FUNCTION_BLOCK FB_SlaveRobot
VAR_INPUT
END_VAR
VAR_OUTPUT
END_VAR
VAR
	// flag if robot self-check passed
	m_selfCheckPass :ARRAY[1..g_sArmNum] OF BOOL :=[4(false)];
	
	// flag if master are connected
	m_masterOnLine :BOOL :=FALSE;
	m_masterOnLineCheck :FB_masterConnectionCheck;
	
	// master-slave motion scale
	m_motionScale :LREAL;
	
	// index(0 to 4) of slave arm which is tele-linked to master arm
	m_teleSlaveArmIdx :ARRAY[1..g_mArmNum] OF E_MatchedSlaveArmIdx;
	
	// flag if endoscope is mounted
	m_endoscopeMounted :BOOL := FALSE;
	
	// endoscope pose in cart coordinate
	m_endoscopePose : ST_Frame;
	
	// endoscope type 
	m_endoscopeType : E_EndoscopeType:= EndoScopeType_30;
	m_lastEndoScopePostureRobot : E_EndoscopePosture:= EndoScopePosture_HeadDown;
	m_lastEndoScopePostureUI : E_EndoscopePosture:= EndoScopePosture_HeadDown;
	
	// slave arms, responsible for arm kinematic and control
	m_slaveArms :ARRAY[1..g_sArmNum] OF FB_SlaveArm;
	
	// arm state
	m_slaveArmState:ARRAY[1..g_sArmNum] OF E_SlaveArmState:=[4(E_SlaveArmState.SlaveArmState_Error)];
	m_lastSlaveArmState:ARRAY[1..g_sArmNum] OF E_SlaveArmState:=[4(E_SlaveArmState.SlaveArmState_Error)];
	m_nextSlaveArmState:ARRAY[1..g_sArmNum] OF E_SlaveArmState:=[4(E_SlaveArmState.SlaveArmState_Error)];
	
	// matched master arm state
	m_matchedMasterArmState :ARRAY[1..g_sArmNum] OF E_MasterArmState:=[4(E_MasterArmState.MasterArmState_Error)];
	
	// flag if panel and instrument mounted
	m_panelMountedFlag :ARRAY[1..g_sArmNum] OF BOOL :=[4(FALSE)];
	m_instrumentMountedFlag :ARRAY[1..g_sArmNum] OF BOOL :=[4(FALSE)];
	
	// flag if enable instrument invasion after it mounted
	m_instruInvasionEnableFlag :ARRAY[1..g_sArmNum] OF BOOL :=[4(FALSE)];
	
	// all arm controller instance 
	m_armCtrlFactory :ARRAY[1..g_sArmNum,1..SlaveArmState_totalNum] OF I_SlaveArmCtrl;
	m_armError :ARRAY[1..g_sArmNum] OF FB_SlaveCtrlError;
	m_armInit :ARRAY[1..g_sArmNum] OF FB_SlaveCtrlInit;
	m_armSelfCheck :ARRAY[1..g_sArmNum] OF FB_SlaveCtrlSelfCheck;
	m_armStandBy :ARRAY[1..g_sArmNum] OF FB_SlaveCtrlStandBy;
	m_mountPanel :ARRAY[1..g_sArmNum] OF FB_SlaveCtrlMountPanel;
	m_panelReady :ARRAY[1..g_sArmNum] OF FB_SlaveCtrlPanelReady;
	m_mountInstru :ARRAY[1..g_sArmNum] OF FB_SlaveCtrlMountInstru;
	m_instruReady :ARRAY[1..g_sArmNum] OF FB_SlaveCtrlInstruReady;
	m_armMasterSlave :ARRAY[1..g_sArmNum] OF FB_SlaveCtrlMasterSlave;
	m_scopeReady :ARRAY[1..g_sArmNum] OF FB_SlaveCtrlScopeReady;
	m_armEndoscope :ARRAY[1..g_sArmNum] OF FB_SlaveCtrlEndoscope;
	m_armAdjust :ARRAY[1..g_sArmNum] OF FB_SlaveCtrlAdjust;
	m_armPackage :ARRAY[1..g_sArmNum] OF FB_SlaveCtrlPackage;
	m_armCart :ARRAY[1..g_sArmNum] OF FB_SlaveCtrlCart;
	m_armGraCali :ARRAY[1..g_sArmNum] OF FB_SlaveCtrlGraCali;
	m_armTest :ARRAY[1..g_sArmNum] OF FB_SlaveCtrlTest;
	m_instruRetract :ARRAY[1..g_sArmNum] OF FB_SlaveCtrlInstruRetract;
	m_instruInvasion :ARRAY[1..g_sArmNum] OF FB_SlaveCtrlInstruInvasion;
	m_armDisable :ARRAY[1..g_sArmNum] OF FB_SlaveCtrlDisable;
	m_instruCali :ARRAY[1..g_sArmNum] OF FB_SlaveCtrlInstruCali;
	m_scopeToggle :ARRAY[1..g_sArmNum] OF FB_SlaveCtrlScopeToggle;
	m_Performance :ARRAY[1..g_sArmNum] OF FB_SlaveCtrlPerformance;
	m_armStop :ARRAY[1..g_sArmNum] OF FB_SlaveCtrlStop;
	
	// arm controller interface
	m_armCtrl :ARRAY[1..g_sArmNum] OF I_SlaveArmCtrl;
	m_armCtrlCmds :ARRAY[1..g_sArmNum] OF ST_SlaveArmCtrlCmds;

END_VAR

METHOD PROTECTED controllerTransit : BOOL
VAR_INPUT
END_VAR
VAR
	i:int;
END_VAR
FOR i:=1 TO g_sArmNum DO 
	// Controller transit
	IF m_nextSlaveArmState[i]<> m_slaveArmState[i] THEN
		// reset current controller
		m_armCtrl[i].reset();
		
		// transit to new controller
		m_lastSlaveArmState[i]:=m_slaveArmState[i];
		m_slaveArmState[i]:=m_nextSlaveArmState[i];
		m_armCtrl[i]:=m_armCtrlFactory[i,m_slaveArmState[i]];
		
		// init next controller
		m_armCtrl[i].Init(m_slaveArms[i],m_armCtrlCmds[i]);
		m_slaveArms[i].updateCmds(m_armCtrlCmds[i]);
	END_IF
END_FOR
END_METHOD

METHOD PUBLIC getStatus : BOOL
VAR_IN_OUT
	// slave robot information, including arm status and cartesian data
	r_slaveStatus :ST_SlaveStatus;
	
	// slave robot joint data
	r_slaveJointsData :ST_SlaveJointData;
	
END_VAR

VAR
	i:INT;
END_VAR
r_slaveStatus.m_armState:=m_slaveArmState;
r_slaveStatus.m_endoscopeMounted :=m_endoscopeMounted;
r_slaveStatus.m_endoscopePose :=m_endoscopePose;

FOR i:=1 TO g_sArmNum DO
	r_slaveStatus.m_selfCheckPass[i] := m_selfCheckPass[i];	

	// instrument data
	r_slaveStatus.m_instruStauts[i].m_type:=m_slaveArms[i].instrument.m_instruType;
	r_slaveStatus.m_instruStauts[i].m_ready:=m_instrumentMountedFlag[i];
	r_slaveStatus.m_instruStauts[i].m_fingerAngle:=m_slaveArms[i].curGripAngle;
	r_slaveStatus.m_instruReadErrId[i] := m_slaveArms[i].instrument.onChipData.m_ErrorID;
	r_slaveStatus.m_instruInstallStatus[i] := m_slaveArms[i].instruOn;
	r_slaveStatus.m_instruClampErrId[i] := m_mountInstru[i].instruClampErrId;
	r_slaveStatus.m_panelInstallStatus[i] := m_slaveArms[i].panelOn;
	r_slaveStatus.m_panelClampErrId[i] := m_mountPanel[i].panelClampErrId;
	r_slaveStatus.m_trocarOnFlag[i] := m_slaveArms[i].trocarOn;
	r_slaveStatus.m_masterOnLine := m_masterOnLine;
	// cartesion
	r_slaveStatus.m_curArmPose[i]:=m_slaveArms[i].curCartPose;
	r_slaveStatus.m_simArmPose[i]:=m_slaveArms[i].simCartPose;
	r_slaveStatus.m_masterSlavePoseError[i] := m_armMasterSlave[i].masterSlavePoseErr;
	// joint
	r_slaveJointsData.m_curMotorPos[i]:=m_slaveArms[i].curMotorPos;
	r_slaveJointsData.m_curLinkPos[i]:=m_slaveArms[i].curLinkPos;
	r_slaveJointsData.m_curJntPos[i]:=m_slaveArms[i].curJntPos;
	r_slaveJointsData.m_curJntVel[i]:=m_slaveArms[i].curJntVel;
	r_slaveJointsData.m_rawJntCurrent[i] := m_slaveArms[i].rawJntCurrent;
	// command info
	// cartesion
	r_slaveStatus.m_cmdArmPose[i]:=m_slaveArms[i].cmdCartPose;
	// joint info
	r_slaveJointsData.m_cmdJntPos[i]:=m_slaveArms[i].cmdJntPos;
	
END_FOR
END_METHOD

METHOD PUBLIC Init : BOOL
VAR_INPUT
END_VAR
VAR
	i:INT;
END_VAR
FOR i:=1 TO g_sArmNum DO
	// arm init
	m_slaveArms[i].Init(i);
	m_slaveArmState[i]:=SlaveArmState_Init;
	m_lastSlaveArmState[i]:=SlaveArmState_Init;
	m_nextSlaveArmState[i]:=SlaveArmState_Init;
	m_selfCheckPass[i]:=false;
	
	// command init
	m_armCtrlCmds[i].m_jntEnableFlag := g_zeroVec8i;
	m_armCtrlCmds[i].m_jntOPMode := g_slaveAllPosMode;
	m_armCtrlCmds[i].m_cmdCartPose := m_slaveArms[i].curCartPose;
	m_armCtrlCmds[i].m_cmdCartTwist := g_zeroVec6d;
	m_armCtrlCmds[i].m_cmdJntPos := m_slaveArms[i].curJntPos;
	m_armCtrlCmds[i].m_cmdJntVel := g_zeroVec8d;
	m_armCtrlCmds[i].m_cmdJntAcc := g_zeroVec8d;
	m_armCtrlCmds[i].m_cmdJntTrq := g_zeroVec8d;
	
	// generate controller factory
	m_armCtrlFactory[i,SlaveArmState_Error] := m_armError[i];
	m_armCtrlFactory[i,SlaveArmState_Init] := m_armInit[i];
	m_armCtrlFactory[i,SlaveArmState_SelfCheck] := m_armSelfCheck[i];
	m_armCtrlFactory[i,SlaveArmState_Standby] := m_armStandBy[i];
	m_armCtrlFactory[i,SlaveArmState_MountPanel] := m_mountPanel[i];
	m_armCtrlFactory[i,SlaveArmState_PanelReady] := m_panelReady[i];
	m_armCtrlFactory[i,SlaveArmState_MountInstru] := m_mountInstru[i];
	m_armCtrlFactory[i,SlaveArmState_InstruReady] := m_instruReady[i];
	m_armCtrlFactory[i,SlaveArmState_MasterSlave] := m_armMasterSlave[i];
	m_armCtrlFactory[i,SlaveArmState_ScopeReady] := m_scopeReady[i];
	m_armCtrlFactory[i,SlaveArmState_EndoScope] := m_armEndoscope[i];
	m_armCtrlFactory[i,SlaveArmState_Adjust] := m_armAdjust[i];
	m_armCtrlFactory[i,SlaveArmState_Package] := m_armPackage[i];
	m_armCtrlFactory[i,SlaveArmState_Cart] := m_armCart[i];
	m_armCtrlFactory[i,SlaveArmState_GravityCali] := m_armGraCali[i];
	m_armCtrlFactory[i,SlaveArmState_Test] := m_armTest[i];
	m_armCtrlFactory[i,SlaveArmState_InstruRetract] := m_instruRetract[i];
	m_armCtrlFactory[i,SlaveArmState_InstruInvasion] := m_instruInvasion[i];
	m_armCtrlFactory[i,SlaveArmState_Disable] := m_armDisable[i];
	m_armCtrlFactory[i,SlaveArmState_InstruCali] := m_instruCali[i];
	m_armCtrlFactory[i,SlaveArmState_ScopeToggle] := m_scopeToggle[i];
	m_armCtrlFactory[i,SlaveArmState_Performance] := m_Performance[i];
	m_armCtrlFactory[i,SlaveArmState_Stop] := m_armStop[i];
	
	// assign controller
	m_armCtrl[i]:=m_armCtrlFactory[i,m_slaveArmState[i]];
	m_armCtrl[i].Init(m_slaveArms[i],m_armCtrlCmds[i]);
END_FOR
END_METHOD

METHOD PUBLIC run : BOOL
VAR_IN_OUT CONSTANT
	i_slaveInputDataPool:ST_SlaveInputDataPool;
END_VAR
VAR
	i:INT;
END_VAR
m_motionScale := i_slaveInputDataPool.m_masterStatus.m_motionScale;
m_teleSlaveArmIdx := i_slaveInputDataPool.m_masterStatus.m_teleSlaveArmIdx;

// check master connection
m_masterOnLine := m_masterOnLineCheck.check(i_slaveInputDataPool.m_masterStatus.m_masterHeartBeat);

// check if endoscope is mounted
m_endoscopeMounted := FALSE;
FOR i:=1 TO g_sArmNum DO 
	IF m_slaveArms[i].instrument.m_instruType=InstruType_endoscope THEN
		m_endoscopeMounted := TRUE;
		m_endoscopePose := transform(i_slaveInputDataPool.m_setupStatus.m_curEndPose[i], m_slaveArms[i].curCartPose);
		m_endoScopeType := m_slaveArms[i].instrument.curScopeType;
		
		//set endoscope  posture from UI data
		updateScopeUIInfo();
	END_IF
END_FOR

// update arm status
FOR i:=1 TO g_sArmNum DO
	// update dynamic data
	m_slaveArms[i].updateDyna(i_slaveInputDataPool.m_slaveDynaData);
								
	// update slave arm kinematics
	m_slaveArms[i].updateStatus();
END_FOR

// state machine transition
stateMachine(i_slaveInputDataPool);

// controller transition
controllerTransit();

// run arm controller
FOR i:=1 TO g_sArmNum DO
	// null ptr check
	ASSERT(0 <> m_armCtrl[i]);
	
	// run controller
	m_armCtrl[i].run(m_endoscopePose, i_slaveInputDataPool.m_MasterStatus,
					i_slaveInputDataPool.m_setupStatus, m_SlaveArms[i],m_armCtrlCmds[i]);

	// update commands to drivers
	m_slaveArms[i].updateCmds(m_armCtrlCmds[i]);
END_FOR
END_METHOD

// state machine check and transit 
METHOD PROTECTED stateMachine : BOOL
VAR_IN_OUT CONSTANT
		i_slavesInputDataPool:ST_SlaveInputDataPool;
END_VAR
VAR
	i,j:INT;
END_VAR
// check instrument state
FOR i:=1 TO g_sArmNum DO
	// statues check
	IF m_slaveArms[i].panelOn = FALSE THEN
		m_panelMountedFlag[i]:=FALSE;
	END_IF
	IF m_slaveArms[i].instruOn = FALSE THEN
		m_instrumentMountedFlag[i]:=FALSE;			
	END_IF
END_FOR

// get matched master arm state
FOR i:=1 TO g_sArmNum DO 
	m_matchedMasterArmState[i]:=MasterArmState_Error;
	FOR j:=1 TO g_mArmNum DO 
		IF i = i_slavesInputDataPool.m_masterStatus.m_teleSlaveArmIdx[j] THEN
			m_matchedMasterArmState[i] := i_slavesInputDataPool.m_masterStatus.m_armState[j];
		END_IF
	END_FOR
END_FOR

// check if to enable instrument invasion 
FOR i:=1 TO g_sArmNum DO
	IF SlaveArmState_Adjust = m_slaveArmState[i] OR SlaveArmState_Cart = m_slaveArmState[i] OR i_slavesInputDataPool.m_setupStatus.m_armState[i] = SetupArmState_ManualAdjust OR
	    m_slaveArms[i].instrument.instruType = InstruType_Endoscope	 THEN
		m_instruInvasionEnableFlag[i]:=FALSE;
		m_slaveArms[i].resetInstruDepth();
	ELSIF m_instrumentMountedFlag[i] AND m_slaveArms[i].instrument.instruType <> InstruType_Endoscope AND m_slaveArmState[i] <> SlaveArmState_InstruInvasion THEN
		m_instruInvasionEnableFlag[i]:=TRUE;
		m_slaveArms[i].setInstruDepth();
	END_IF
END_FOR  

// state machine transit
FOR i:=1 TO g_sArmNum DO
	CASE m_slaveArmState[i] OF
		// error
		SlaveArmState_Error:
			IF FALSE = i_slavesInputDataPool.m_safetyData.m_slaveErrFlag[i] THEN
				// to standby
				IF m_selfCheckPass[i] THEN
					m_nextSlaveArmState[i] :=SlaveArmState_Standby;
				// to init
				ELSE
					m_nextSlaveArmState[i] :=SlaveArmState_Init;
				END_IF
			END_IF
			// to adjust
			IF (m_slaveArms[i].adjustOn) THEN
				m_nextSlaveArmState[i]:=SlaveArmState_Adjust;
			END_IF
			
		// init
		SlaveArmState_Init:
			m_selfCheckPass[i]:=FALSE;
			m_slaveArms[i].instrument.resetArmLED :=TRUE;
			// to selfcheck
			IF m_armCtrl[i].isFinished AND i_slavesInputDataPool.m_masterStatus.m_slaveSelfCheckFlag  THEN
				m_nextSlaveArmState[i]:=SlaveArmState_SelfCheck;
			// to adjust
			ELSIF m_slaveArms[i].adjustOn THEN
				m_nextSlaveArmState[i]:=SlaveArmState_Adjust;
			END_IF

		//self check
		SlaveArmState_SelfCheck:
			// to standby
			IF m_armCtrl[i].isFinished  THEN
				m_nextSlaveArmState[i]:=SlaveArmState_Standby;
				m_selfCheckPass[i]:=TRUE;
			END_IF
		
		//standby
		SlaveArmState_Standby:
			// to mount panel
			IF m_slaveArms[i].panelOn THEN 
				IF m_panelMountedFlag[i] THEN
					m_nextSlaveArmState[i]:=SlaveArmState_PanelReady;
				ELSE
					m_nextSlaveArmState[i]:=SlaveArmState_MountPanel;
				END_IF
			// to adjust
			ELSIF m_slaveArms[i].adjustOn THEN
				m_nextSlaveArmState[i]:=SlaveArmState_Adjust;
			END_IF
		
		//mount panel
		SlaveArmState_MountPanel:
			// to panel ready
			IF m_armCtrl[i]. isFinished THEN
				m_nextSlaveArmState[i]:=SlaveArmState_PanelReady;
				m_panelMountedFlag[i] :=TRUE;
				
			// to standby
			ELSIF NOT(m_slaveArms[i].panelOn) THEN
				m_nextSlaveArmState[i]:=SlaveArmState_Standby;
			END_IF
		
		//panel ready
		SlaveArmState_PanelReady:
			// to adjust
			IF (m_slaveArms[i].adjustOn) THEN
				m_nextSlaveArmState[i]:=SlaveArmState_Adjust;
			// to stand by
			ELSIF NOT(m_slaveArms[i].panelOn) THEN
				m_nextSlaveArmState[i]:=SlaveArmState_Standby;
			ELSIF m_slaveArms[i].instruOn   THEN
				IF m_instrumentMountedFlag[i] THEN
					// to scope ready
					IF  InstruType_endoscope = m_slaveArms[i].instrument.m_instruType AND m_slaveArms[i].instruReady() THEN 
						m_nextSlaveArmState[i]:=SlaveArmState_ScopeReady;
					// to scope toggle
					ELSIF  InstruType_endoscope = m_slaveArms[i].instrument.m_instruType AND 
								(m_slaveArms[i].instrument.curScopePosture <> m_slaveArms[i].instrument.nextScopePosture OR
								m_slaveArms[i].instrument.curScopeType <> m_slaveArms[i].instrument.nextScopeType) THEN
						m_nextSlaveArmState[i] := SlaveArmState_ScopeToggle;
					// to instrument ready
					ELSIF  m_slaveArms[i].instruReady() THEN
						m_nextSlaveArmState[i]:=SlaveArmState_InstruReady;
					END_IF
				// to mount instrument/endoscope
				ELSIF m_slaveArms[i].readyForInstruMount() THEN
					m_nextSlaveArmState[i]:=SlaveArmState_MountInstru;
				END_IF
			// to instrument retract
			ELSIF  NOT(m_slaveArms[i].readyForInstruMount())  THEN
				m_nextSlaveArmState[i]:=SlaveArmState_InstruRetract;
			END_IF
			
		//mount instrument
		SlaveArmState_MountInstru:
			// to panel ready
			IF NOT(m_slaveArms[i].instruOn)  THEN
				m_nextSlaveArmState[i]:=SlaveArmState_PanelReady;
			ELSIF m_armCtrl[i].isFinished THEN
				m_instrumentMountedFlag[i] :=TRUE;
				
				// to instrument invasion
				IF m_instruInvasionEnableFlag[i] THEN
					m_nextSlaveArmState[i] := SlaveArmState_InstruInvasion;
				// to panel ready
				ELSE
					m_nextSlaveArmState[i]:=SlaveArmState_PanelReady;
				END_IF
				
			END_IF
		
		// instrument ready
		SlaveArmState_InstruReady:
			// to instrument retract
			IF  NOT(m_slaveArms[i].instruOn)  THEN
				m_nextSlaveArmState[i]:=SlaveArmState_InstruRetract;
			// to Adjust
			ELSIF (m_slaveArms[i].adjustOn) THEN
				m_nextSlaveArmState[i]:=SlaveArmState_Adjust;
			// to master-slave
			ELSIF MasterArmState_MasterSlave = m_matchedMasterArmState[i] THEN
				m_nextSlaveArmState[i] := SlaveArmState_MasterSlave;
			END_IF
		
		//master slave control
		SlaveArmState_MasterSlave:
			// to Adjust
			IF (m_slaveArms[i].adjustOn) THEN
				m_nextSlaveArmState[i]:=SlaveArmState_Adjust;
			// to stop
			ELSIF MasterArmState_MasterSlave <> m_matchedMasterArmState[i] OR m_armCtrl[i].isFinished THEN
				m_nextSlaveArmState[i]:=SlaveArmState_Stop;
				m_armStop[i].setInstruBacklash(m_armMasterSlave[i].InstruBacklash);
			// to instrument retract
			ELSIF  NOT(m_slaveArms[i].panelOn) OR NOT(m_slaveArms[i].instruOn) THEN
				m_nextSlaveArmState[i]:=SlaveArmState_InstruRetract;
			END_IF
		
		//endoscope ready
		SlaveArmState_ScopeReady:
			// to instrument retract
			IF NOT(m_slaveArms[i].instruOn) THEN
				m_nextSlaveArmState[i]:=SlaveArmState_InstruRetract;
			// to Adjust
			ELSIF (m_slaveArms[i].adjustOn) THEN
				m_nextSlaveArmState[i]:=SlaveArmState_Adjust;
			// to scope toggle
			ELSIF m_slaveArms[i].instrument.curScopePosture <> m_slaveArms[i].instrument.nextScopePosture OR
					m_slaveArms[i].instrument.curScopeType <> m_slaveArms[i].instrument.nextScopeType THEN
				m_nextSlaveArmState[i] := SlaveArmState_ScopeToggle;
			// to endoscope control
			ELSIF MasterArmState_Endoscope = i_slavesInputDataPool.m_masterStatus.m_armState[1] AND 
				  MasterArmState_Endoscope = i_slavesInputDataPool.m_masterStatus.m_armState[2] THEN
				m_nextSlaveArmState[i] := SlaveArmState_EndoScope;
			END_IF
		
		//endoscope control
		SlaveArmState_EndoScope:
			// to Adjust
			IF (m_slaveArms[i].adjustOn) THEN
				m_nextSlaveArmState[i]:=SlaveArmState_Adjust;
			// to stop
			ELSIF MasterArmState_Endoscope <> i_slavesInputDataPool.m_masterStatus.m_armState[1]
				OR MasterArmState_Endoscope <> i_slavesInputDataPool.m_masterStatus.m_armState[2] THEN
				m_nextSlaveArmState[i]:=SlaveArmState_Stop;
			// to scope toggle
			ELSIF m_slaveArms[i].instrument.curScopePosture <> m_slaveArms[i].instrument.nextScopePosture OR
					m_slaveArms[i].instrument.curScopeType <> m_slaveArms[i].instrument.nextScopeType THEN
				m_nextSlaveArmState[i] := SlaveArmState_ScopeToggle;
			// to instrument retract
			ELSIF  NOT(m_slaveArms[i].panelOn) OR NOT(m_slaveArms[i].instruOn) THEN
				m_nextSlaveArmState[i]:=SlaveArmState_InstruRetract;
			END_IF
			
		//arm adjust
		SlaveArmState_Adjust:
			IF m_slaveArms[i].adjustFallEdge AND m_armCtrl[i].timePeriod > 0.25 THEN
				// to init
				IF NOT (m_selfCheckPass[i]) THEN
					m_nextSlaveArmState[i] :=SlaveArmState_Init;
				// to standby
				ELSE
					m_nextSlaveArmState[i] :=SlaveArmState_Standby;
				END_IF
			END_IF
		
		//scope toggle
		SlaveArmState_ScopeToggle:
			// to instrument retract
			IF NOT(m_slaveArms[i].instruOn) THEN
				m_nextSlaveArmState[i]:=SlaveArmState_InstruRetract;
			// to standby
			ELSIF m_armCtrl[i].isFinished THEN
				m_nextSlaveArmState[i] :=SlaveArmState_Standby;
			END_IF
		
		// package
		SlaveArmState_Package:
			// to Adjust
			IF (m_slaveArms[i].adjustOn) THEN
				m_nextSlaveArmState[i]:=SlaveArmState_Adjust;
			// to standby
			ELSIF m_armCtrl[i].isFinished THEN
				m_nextSlaveArmState[i]:=SlaveArmState_Standby;
			END_IF
			
		// Cart
		SlaveArmState_Cart:
		
		// Gravity Calibration
		SlaveArmState_GravityCali:
			// to Adjust
			IF (m_slaveArms[i].adjustOn) THEN
				m_nextSlaveArmState[i]:=SlaveArmState_Adjust;
			// to standby
			ELSIF m_armCtrl[i].isFinished THEN
				m_nextSlaveArmState[i]:=SlaveArmState_Standby;
			END_IF
			
		//arm test
		SlaveArmState_Test:
			// to stop
			IF  m_armCtrl[i].isFinished THEN
				m_nextSlaveArmState[i]:=SlaveArmState_Stop;
			END_IF
		
		//arm Performance
		SlaveArmState_Performance:
			// to standby
			IF  m_armCtrl[i].isFinished THEN
				m_nextSlaveArmState[i]:=SlaveArmState_Standby;
			END_IF		
			
		//arm stop
		SlaveArmState_Stop:
			// to standby
			IF  m_armCtrl[i].isFinished THEN
				m_nextSlaveArmState[i]:=SlaveArmState_Standby;
			END_IF
		
		// instrument retract
		SlaveArmState_InstruRetract:
			// to Adjust
			IF (m_slaveArms[i].adjustOn) THEN
				m_nextSlaveArmState[i]:=SlaveArmState_Adjust;
			// to standby
			ELSIF m_armCtrl[i].isFinished THEN
				m_nextSlaveArmState[i]:=SlaveArmState_Standby;
			END_IF
		
		// instrument invasion
		SlaveArmState_InstruInvasion:
			// to instrument retract
			IF NOT m_slaveArms[i].instruOn THEN
				m_nextSlaveArmState[i]:=SlaveArmState_InstruRetract;
			// to Adjust
			elsIF (m_slaveArms[i].adjustOn) THEN
				m_nextSlaveArmState[i]:=SlaveArmState_Adjust;
			// to instrument ready
			ELSIF m_armCtrl[i].isFinished THEN
			// to panel ready
				m_nextSlaveArmState[i]:=SlaveArmState_PanelReady;
			END_IF
		
		// arm disable
		SlaveArmState_Disable:
			IF NOT(i_slavesInputDataPool.m_UIData.m_slaveArmDisableFlag[i]) THEN
				// to standby
				IF m_selfCheckPass[i] THEN
					m_nextSlaveArmState[i] :=SlaveArmState_Standby;
				// to init
				ELSE
					m_nextSlaveArmState[i] :=SlaveArmState_Init;
				END_IF
			END_IF
	END_CASE
	
	// control is forbidden if setup arm is not in Hold
	IF SetupArmState_Hold <> i_slavesInputDataPool.m_setupStatus.m_armState[i] AND
		(SlaveArmState_InstruReady = m_nextSlaveArmState[i] OR SlaveArmState_MasterSlave = m_nextSlaveArmState[i]
		 OR SlaveArmState_ScopeReady = m_nextSlaveArmState[i] OR SlaveArmState_EndoScope = m_nextSlaveArmState[i]) THEN
		m_nextSlaveArmState[i]:=SlaveArmState_Standby;
	END_IF
	
	// arm disable
	IF i_slavesInputDataPool.m_UIData.m_slaveArmDisableFlag[i] THEN
		m_nextSlaveArmState[i] := SlaveArmState_Disable;
	// error check
	ELSIF i_slavesInputDataPool.m_safetyData.m_slaveErrFlag[i] AND NOT m_slaveArms[i].adjustOn THEN
		m_nextSlaveArmState[i]:=SlaveArmState_Error;
	END_IF
END_FOR
END_METHOD

METHOD PROTECTED updateScopeUIInfo : BOOL
VAR_INPUT
END_VAR
VAR
	i:INT;
END_VAR
// check if endoscope is mounted
FOR i:=1 TO g_sArmNum DO 
	IF m_slaveArms[i].instrument.m_instruType=InstruType_endoscope THEN
		
		// update command endoscope posture from UI
		IF GVL_interactUI.g_scopeUpDown <> m_lastEndoScopePostureUI AND m_slaveArms[i].instrument.curScopeType = EndoScopeType_30 THEN
			IF GVL_interactUI.g_scopeUpDown = 1 THEN
				m_slaveArms[i].instrument.nextScopePosture := EndoScopePosture_HeadDown;
			ELSIF  GVL_interactUI.g_scopeUpDown = 2 THEN
				m_slaveArms[i].instrument.nextScopePosture := EndoscopePosture_HeadUp;
			END_IF
		END_IF
		
		// update current endoscope posture to UI
		IF m_slaveArms[i].instrument.curScopePosture <> m_lastEndoScopePostureRobot THEN
			IF m_slaveArms[i].instrument.curScopePosture = EndoScopePosture_HeadDown THEN
				GVL_interactUI.g_scopeUpDown := 1 ;
			ELSIF  m_slaveArms[i].instrument.curScopePosture = EndoScopePosture_HeadUp THEN
				GVL_interactUI.g_scopeUpDown := 2;
			END_IF
		END_IF
		m_lastEndoScopePostureRobot := m_slaveArms[i].instrument.curScopePosture;
		
	END_IF
END_FOR

m_lastEndoScopePostureUI := GVL_interactUI.g_scopeUpDown;
END_METHOD

END_FUNCTION_BLOCK

(* stored: Version 1.1.0.1, ProductVersion 3.1.4024.11
   POU FB_SlaveRobot: Id {8cbdb2ba-9735-46e3-8cbc-296330acc8cc}, SpecialFunc None
   Method controllerTransit: Id {8f288ee3-c1dd-4604-a493-d121fbcd6b66}
   Method getStatus: Id {b6139e8c-2703-424c-9761-ad1add6b1ff1}
   Method Init: Id {610a17f3-34c5-4e3c-bbbc-19f9c2f46946}
   Method run: Id {ed6f787a-4dc0-4602-b386-92a3c3880a23}
   Method stateMachine: Id {b9cc8560-9309-49e3-93b5-28cb02b4f5cc}
   Method updateScopeUIInfo: Id {8acce6ed-98d8-433e-be8e-5c90fe998877} *)
